TYPE OutputBase_10CEE7DE :
STRUCT
END_STRUCT
END_TYPE

(* stored: Version 1.2.0.0
   DUT OutputBase_10CEE7DE: Id {431f079d-2b68-49ef-a125-646bfa2b031b} *)
